	                #sFB_RightAngledTransfer_541(iUDT_Configuration := #iUDT_Configuration."541".RightAngledTransfer,
	                                             iUDT_LowerConveyorConfiguration := #iUDT_Configuration."540".Conveyor,
	                                             iUDT_UpperConveyorConfiguration := #iUDT_Configuration."541".Conveyor,
	                                             iUDT_PECConfiguration := #iUDT_Configuration."540".PEC,
	                                             ii_DestinationA := #si_540DestinationA,
	                                             ii_DestinationB := #si_540DestinationB,
	                                             ii_DestinationC := #si_540DestinationC,
	                                             ii_DestinationD := #si_540DestinationD,
	                                             ix_HardwareOk := #ix_HardwareOk,
	                                             ix_400vOk := #ix_400vOk,
	                                             ix_24vOk := #ix_24vOk,
	                                             ix_SafetyOk := #ix_SafetyOk,
	                                             ix_AirPressureOk := #ix_AirPressureOk,
	                                             ix_SectionIsDown := #ix_SectionIsDown541,
	                                             ix_SectionIsUp := #ix_SectionIsUp541,
	                                             ix_ConveyorAAuto := #iqUDT_WorkstationCommonStatus."530".AutoON,
	                                             ix_ConveyorBAuto := #iqUDT_WorkstationCommonStatus."550".AutoON,
	                                             ix_ConveyorCAuto := #iqUDT_WorkstationCommonStatus."670".AutoON,
	                                             ix_ConveyorDAuto := FALSE,
	                                             ix_PEC := #iUDT_MotorInput540.AllSensorPortInputs.LeftSensor,
	                                             ix_ExternalReceiveRequestA := NOT #iqUDT_WorkstationStatus."530".PEC_Eos.PEC AND NOT #sx_TransferOut380 AND NOT #sx_TransferOut390,
	                                             ix_ExternalReceiveRequestB := false,
	                                             ix_ExternalReceiveRequestC := #sFB_RightAngledTransfer_671.qx_ExternalSendRequestC,
	                                             ix_ExternalReceiveRequestD := false,
	                                             ix_PECInfeedA := #iqUDT_WorkstationStatus."530".PEC_Eos.PEC,
	                                             ix_PECInfeedC := #iqUDT_WorkstationStatus."670".PEC_Eos.PEC,
	                                             qUDT_HMIRATStatus => #iqUDT_WorkstationStatus."541".RightAngledTransfer,
	                                             qUDT_HMIConveyorStatus => #iqUDT_WorkstationStatus."540".Conveyor,
	                                             qUDT_HMIPECStatus => #iqUDT_WorkstationStatus."540".PEC_Eos,
	                                             qUDT_RATStatus => #iqUDT_WorkstationCommonStatus."541",
	                                             qUDT_ConveyorStatus => #iqUDT_WorkstationCommonStatus."540",
	                                             qx_PopupControl => #qx_PopupControl541,
	                                             iqUDT_EquipmentControl := #iqUDT_EquipmentControl,
	                                             iqUDT_RATCommand := #iqUDT_WorkstationCommands."541".RightAngledTransfer,
	                                             iqUDT_ConveyorCommand := #iqUDT_WorkstationCommands."540".Conveyor,
	                                             iqUDT_RATStatistics := #iqUDT_WorkstationStatistics."541".RightAngledTransfer,
	                                             iqUDT_ConveyorStatistics := #iqUDT_WorkstationStatistics."540".Conveyor,
	                                             iqUDT_PECStatistics := #iqUDT_WorkstationStatistics."540".PEC_Eos,
	                                             iqUDT_HandShakeConveyorA := #sUDT_Handshake_530,
	                                             iqUDT_HandShakeConveyorB := #sUDT_Handshake_540,
	                                             iqUDT_HandShakeConveyorC := #sUDT_HandshakeUp_671,
	                                             iqUDT_HandShakeConveyorD := #tUDT_dummyHandshake,
	                                             iqUDT_LowerConveyorInterface := #sUDT_Interface_540,
	                                             iqUDT_UpperConveyorInterface := #sUDT_Interface_541,
	                                             iqUDT_RATPositioning := #iqUDT_RATPositioning540,
	                                             iqUDT_BladeStopEoSInterface := #tUDT_DummyBladeStop,
	                                             iqUDT_BladeStopBoSInterface := #tUDT_DummyBladeStop);

	            END_REGION

	            REGION MCO
	                #sFB_MCOConveyLinxAixController_541(iUDT_AixConfig := #iUDT_Configuration."541".MCO_M01,
	                                                    iv_AixInputsModule := #iUDT_MotorInput540,
	                                                    ii_PositionSetpoint := #iqUDT_RATPositioning540.Upper.EndPosition,
	                                                    ix_24vOk := #ix_24vOk,
	                                                    ix_SimulationModeActive := "DB_Memory".Simulation,
	                                                    ii_MotorPositionId := 2,
	                                                    ix_StartPositioning := #iqUDT_RATPositioning540.Upper.Start,
	                                                    ix_ResetPosition := #iqUDT_RATPositioning540.Upper.ResetPosition,
	                                                    qUDT_HMIStatus => #iqUDT_WorkstationStatus."541".MCO_M01,
	                                                    qx_Positioned => #iqUDT_RATPositioning540.Upper.Done,
	                                                    iqv_AixOutputsModule := #qUDT_MotorOutput540,
	                                                    iqUDT_ConveyorInterface := #sUDT_Interface_541,
	                                                    iqUDT_MCOStatistics := #iqUDT_WorkstationStatistics."541".MCO_M01);
	            END_REGION

	        END_REGION

	        REGION 550

	            REGION Displacement

	                #sFB_Displacement550(#sUDT_Interface_550);

	            END_REGION

	            REGION Tracking

	                #sFB_Tracking_550(iUDT_ConveyorCommonConfiguration := #iUDT_Configuration."550".Conveyor.Common,
	                                  iqa_TrackingData := #sa_TrackingArray_550,
	                                  iqUDT_ConveyorInterface := #sUDT_Interface_550,
	                                  iqUDT_HandshakeUp := #sUDT_Handshake_540,
	                                  iqUDT_Handshake := #sUDT_Handshake_550);
	            END_REGION

	            REGION EOS

	                #sFB_PECUpdate_550(iUDT_PECUpdateConfiguration := #iUDT_Configuration."550".PEC_EoS,
	                                   iUDT_ConveyorCommonConfiguration := #iUDT_Configuration."550".Conveyor.Common,
	                                   ix_PEC := #iUDT_MotorInput550.AllSensorPortInputs.LeftSensor,
	                                   ix_TeachingMode := FALSE,
	                                   qUDT_Status => #iqUDT_WorkstationStatus."550".PEC_EoS,
	                                   qi_GINwrite => #ti_dummy,
	                                   qx_PECFiltered => #tx_dummy,
	                                   iqa_TrackingData := #sa_TrackingArray_550,
	                                   iqUDT_ConveyorInterface := #sUDT_Interface_550,
	                                   iqUDT_UnknownGINRange := #iqUDT_UnknownGINRange,
	                                   iqUDT_FifoHeader := "DB_FIFOLostGIN".Header,
	                                   iqa_FifoData := "DB_FIFOLostGIN".Data,
	                                   iqUDT_Statistics := #iqUDT_WorkstationStatistics."550".PEC_EoS);

	            END_REGION

	            REGION Conveyor
	                #sFB_Conveyor_550(iUDT_ConveyorConfiguration := #iUDT_Configuration."550".Conveyor,
	                                  idi_PECEoSDistance := #iUDT_Configuration."550".PEC_EoS.Distance,
	                                  idi_PECBoSDistance := 0,
	                                  ii_ExternalSpeed := 0,
	                                  ix_SafetyOk := #ix_SafetyOk,
	                                  ix_24vOk := #ix_24vOk,
	                                  ix_400vOk := #ix_400vOk,
	                                  ix_HardwareOk := #ix_HardwareOk,
	                                  ix_PECEoS := #iqUDT_WorkstationStatus."550".PEC_EoS.PEC,
	                                  ix_PECBoS := TRUE,
	                                  ix_ExternalRequestHold := false,
	                                  qUDT_HMIStatus => #iqUDT_WorkstationStatus."550".Conveyor,
	                                  qUDT_Status => #iqUDT_WorkstationCommonStatus."550",
	                                  iqUDT_EquipmentControl := #iqUDT_EquipmentControl,
	                                  iqUDT_ConveyorCommand := #iqUDT_WorkstationCommands."550".Conveyor,
	                                  iqUDT_ConveyorInterface := #sUDT_Interface_550,
	                                  iqUDT_HandShakeUp := #sUDT_Handshake_540,
	                                  iqUDT_HandShake := #sUDT_Handshake_550,
	                                  iqUDT_Statistics := #iqUDT_WorkstationStatistics."550".Conveyor);
	            END_REGION

	            REGION MCO
	                #sFB_MCOConveyLinxAixController_550(iUDT_AixConfig := #iUDT_Configuration."550".MCO_M01,
	                                                    iv_AixInputsModule := #iUDT_MotorInput550,
	                                                    ix_24vOk := #ix_24vOk,
	                                                    ix_SimulationModeActive := "DB_Memory".Simulation,
	                                                    ii_MotorPositionId := 1,
	                                                    qUDT_HMIStatus => #iqUDT_WorkstationStatus."550".MCO_M01,
	                                                    iqv_AixOutputsModule := #qUDT_MotorOutput550,
	                                                    iqUDT_ConveyorInterface := #sUDT_Interface_550,
	                                                    iqUDT_MCOStatistics := #iqUDT_WorkstationStatistics."550".MCO_M01);
	            END_REGION
	        END_REGION

	        REGION 560


	            REGION Displacement

	                #sFB_Displacement560(#sUDT_Interface_560);

	            END_REGION

	            REGION Conveyor
	                #sFB_Conveyor_560(iUDT_ConveyorConfiguration := #iUDT_Configuration."560".Conveyor,
	                                  idi_PECEoSDistance := 0,
	                                  idi_PECBoSDistance := 0,
	                                  ii_ExternalSpeed := 0,
	                                  ix_SafetyOk := #ix_SafetyOk,
	                                  ix_24vOk := #ix_24vOk,
	                                  ix_400vOk := #ix_400vOk,
	                                  ix_HardwareOk := #ix_HardwareOk,
	                                  ix_PECEoS := TRUE,
	                                  ix_PECBoS := TRUE,
	                                  ix_ExternalRequestHold := false,
	                                  qUDT_HMIStatus => #iqUDT_WorkstationStatus."560".Conveyor,
	                                  qUDT_Status => #iqUDT_WorkstationCommonStatus."560",
	                                  iqUDT_EquipmentControl := #iqUDT_EquipmentControl,
	                                  iqUDT_ConveyorCommand := #iqUDT_WorkstationCommands."560".Conveyor,
	                                  iqUDT_ConveyorInterface := #sUDT_Interface_560,
	                                  iqUDT_HandShakeUp := #sUDT_Handshake_550,
	                                  iqUDT_HandShake := #sUDT_Handshake_560,
	                                  iqUDT_Statistics := #iqUDT_WorkstationStatistics."560".Conveyor);
	            END_REGION

	            REGION VFD

	                #sFB_VfdNORDPPO4_560(iUDT_VFDConfig := #iUDT_Configuration."560".VFD,
	                                     iUDT_VFDInputs := #iUDT_MotorInput560,
	                                     iUDT_MotorData := #iUDT_MotorData560,
	                                     ix_24vOk := #ix_24vOk,
	                                     ix_400vOk := #ix_400vOk,
	                                     ix_QuickStopDisable := TRUE,
	                                     ix_SimulationModeActive := "DB_Memory".Simulation,
	                                     qUDT_HMIStatus => #iqUDT_WorkstationStatus."560".VFD,
	                                     qUDT_VFDOutputs => #qUDT_MotorOutput560,
	                                     iqUDT_ConveyorInterface := #sUDT_Interface_560,
	                                     iqUDT_VFDStatistics := #iqUDT_WorkstationStatistics."560".VFD,
	                                     iqx_StartCommissioning := #iqx_StartComissioning560);

	            END_REGION

	        END_REGION

	        REGION 570

	            REGION Displacement

	                #sFB_Displacement570(#sUDT_Interface_570);

	            END_REGION

	            REGION EoS

	                #sFB_PEC_570(ix_PEC := #iUDT_MotorInput570.AllSensorPortInputs.LeftSensor,
	                             iUDT_PECConfiguration := #iUDT_Configuration."570".PEC_EoS,
	                             qUDT_HMIStatus => #iqUDT_WorkstationStatus."570".PEC_EoS,
	                             iqUDT_ConveyorInterface := #sUDT_Interface_570,
	                             iqUDT_PECStatistics := #iqUDT_WorkstationStatistics."570".PEC_EoS);

	            END_REGION

	            REGION Conveyor
	                #sFB_Conveyor_570(iUDT_ConveyorConfiguration := #iUDT_Configuration."570".Conveyor,
	                                  idi_PECEoSDistance := #iUDT_Configuration."570".PEC_EoS.Distance,
	                                  idi_PECBoSDistance := 0,
	                                  ii_ExternalSpeed := 0,
	                                  ix_SafetyOk := #ix_SafetyOk,
	                                  ix_24vOk := #ix_24vOk,
	                                  ix_400vOk := #ix_400vOk,
	                                  ix_HardwareOk := #ix_HardwareOk,
	                                  ix_PECEoS := #iqUDT_WorkstationStatus."570".PEC_EoS.PEC,
	                                  ix_PECBoS := TRUE,
	                                  ix_ExternalRequestHold := false,
	                                  qUDT_HMIStatus => #iqUDT_WorkstationStatus."570".Conveyor,
	                                  qUDT_Status => #iqUDT_WorkstationCommonStatus."570",
	                                  iqUDT_EquipmentControl := #iqUDT_EquipmentControl,
	                                  iqUDT_ConveyorCommand := #iqUDT_WorkstationCommands."570".Conveyor,
	                                  iqUDT_ConveyorInterface := #sUDT_Interface_570,
	                                  iqUDT_HandShakeUp := #sUDT_Handshake_560,
	                                  iqUDT_HandShake := #sUDT_Handshake_570,
	                                  iqUDT_Statistics := #iqUDT_WorkstationStatistics."570".Conveyor);
	            END_REGION

	            REGION MCO
	                #sFB_MCOConveyLinxAixController_570(iUDT_AixConfig := #iUDT_Configuration."570".MCO_M01,
	                                                    iv_AixInputsModule := #iUDT_MotorInput570,
	                                                    ix_24vOk := #ix_24vOk,
	                                                    ix_SimulationModeActive := "DB_Memory".Simulation,
	                                                    ii_MotorPositionId := 1,
	                                                    qUDT_HMIStatus => #iqUDT_WorkstationStatus."570".MCO_M01,
	                                                    iqv_AixOutputsModule := #qUDT_MotorOutput570,
	                                                    iqUDT_ConveyorInterface := #sUDT_Interface_570,
	                                                    iqUDT_MCOStatistics := #iqUDT_WorkstationStatistics."570".MCO_M01);
	            END_REGION
	        END_REGION

	        REGION 580

	            REGION Displacement

	                #sFB_Displacement580(#sUDT_Interface_580);

	            END_REGION

	            REGION EoS

	                #sFB_PEC_580(ix_PEC := #iUDT_MotorInput570.AllSensorPortInputs.RightSensor,
	                             iUDT_PECConfiguration := #iUDT_Configuration."580".PEC_EoS,
	                             qUDT_HMIStatus => #iqUDT_WorkstationStatus."580".PEC_EoS,
	                             iqUDT_ConveyorInterface := #sUDT_Interface_580,
	                             iqUDT_PECStatistics := #iqUDT_WorkstationStatistics."580".PEC_EoS);

	            END_REGION

	            REGION Conveyor
	                #iqUDT_HandshakeDownstream580.RTR := #iqUDT_HandshakeDownstream580.RTR OR #iqUDT_WorkstationStatus."580".PEC_EoS.PEC;
	                #sFB_Conveyor_580(iUDT_ConveyorConfiguration := #iUDT_Configuration."580".Conveyor,
	                                  idi_PECEoSDistance := #iUDT_Configuration."580".PEC_EoS.Distance,
	                                  idi_PECBoSDistance := 0,
	                                  ii_ExternalSpeed := 0,
	                                  ix_SafetyOk := #ix_SafetyOk,
	                                  ix_24vOk := #ix_24vOk,
	                                  ix_400vOk := #ix_400vOk,
	                                  ix_HardwareOk := #ix_HardwareOk,
	                                  ix_PECEoS := #iqUDT_WorkstationStatus."580".PEC_EoS.PEC,
	                                  ix_PECBoS := TRUE,
	                                  ix_ExternalRequestHold := false,
	                                  qUDT_HMIStatus => #iqUDT_WorkstationStatus."580".Conveyor,
	                                  qUDT_Status => #iqUDT_WorkstationCommonStatus."580",
	                                  iqUDT_EquipmentControl := #iqUDT_EquipmentControl,
	                                  iqUDT_ConveyorCommand := #iqUDT_WorkstationCommands."580".Conveyor,
	                                  iqUDT_ConveyorInterface := #sUDT_Interface_580,
	                                  iqUDT_HandShakeUp := #sUDT_Handshake_570,
	                                  iqUDT_HandShake := #iqUDT_HandshakeDownstream580,
	                                  iqUDT_Statistics := #iqUDT_WorkstationStatistics."580".Conveyor);
	            END_REGION
	            REGION MCO
	                #sFB_MCOConveyLinxAixController_580(iUDT_AixConfig := #iUDT_Configuration."580".MCO_M01,
	                                                    iv_AixInputsModule := #iUDT_MotorInput570,
	                                                    ix_24vOk := #ix_24vOk,
	                                                    ix_SimulationModeActive := "DB_Memory".Simulation,
	                                                    ii_MotorPositionId := 2,
	                                                    qUDT_HMIStatus => #iqUDT_WorkstationStatus."580".MCO_M01,
	                                                    iqv_AixOutputsModule := #qUDT_MotorOutput570,
	                                                    iqUDT_ConveyorInterface := #sUDT_Interface_580,
	                                                    iqUDT_MCOStatistics := #iqUDT_WorkstationStatistics."580".MCO_M01);
	            END_REGION
	        END_REGION
	    END_REGION
	END_IF;


END_FUNCTION_BLOCK

